FUNCTION_BLOCK FB_mbReadSingleReg
VAR_INPUT
	Robot : STRING;
	Register : UINT;
END_VAR
VAR_OUTPUT
	Value : WORD;
END_VAR
VAR
	mbRead : FB_mbReadRegs;
	state : int;
END_VAR

(* 
FB_mbReadSingleReg - Function Block that can be called to read a single MODBUS register from a pre-defined UR Robot
	INPUTS:
		- Robot: 'UR5' or 'UR3'
		- Register: register number to read
	OUTPUTS
		- Value: The returned value
*)

// Set function block vairables
mbRead.nQuantity := 1;
mbRead.cbLength := 2;

IF Robot='UR5' THEN
	mbRead.sIPAddr := Global.stUR5.IP;
	mbRead.nTCPPort := Global.stUR5.mbPort;
	mbRead.nUnitID := Global.stUR5.unitID;
ELSIF Robot='UR3' THEN
	mbRead.sIPAddr := Global.stUR3.IP;
	mbRead.nTCPPort := Global.stUR3.mbPort;
	mbRead.nUnitID := Global.stUR3.unitID;
END_IF

mbRead.pDestAddr := ADR(Value);
mbRead.nMBAddr := Register;

// Set/Determine State of Function block
CASE state OF
	0:
		mbRead.bExecute := TRUE;
		state := 10;
	10:
		IF NOT mbRead.bBusy THEN
			mbRead.bExecute :=FALSE;
			state := 0;
		END_IF
END_CASE

// Run function block
mbRead();

END_FUNCTION_BLOCK

(* stored: Version 1.1.0.1, ProductVersion 3.1.4020.12
   POU FB_mbReadSingleReg: Id {230d1009-9a7b-403f-9bb4-609c9552ea77}, SpecialFunc None *)
